Fanuc KAREL source: IO0072.KL

-- PROVISIONAL review KL for V940-1; original PC SHA256 c1c2a99b13fa0c8d7c35f1b90c9735473d2f50d53c25b610d3cd1d38be079865
-- Incomplete behavior may be omitted. Consult companion uncertainty JSON. Do not deploy.
PROGRAM IO0072
%NOLOCKGROUP
-- UNRESOLVED_LOCAL_POOL 5 cells at code offset 13; source declarations unknown
-- DIRECT_LOCAL_WORD_ACCESS alone does not prove INTEGER, REAL, or BOOLEAN
BEGIN
  -- V9_ZERO_TABLE_METADATA_HINT layout=0001; no indexed target words; source/name/runtime held
  -- V9_ZERO_GLOBAL_LAYOUT_HINT count-one $GROUP table, zero relocation slots, two routine descriptors; executable preamble and source held
  -- V9_ANALOG_RDI_SIGNAL_HINT AIN read I_plus_1
  -- UNRESOLVED_PC offsets 0-18; opcodes 2B,2C,7B
  -- UNRESOLVED_PC offsets 23-30; opcodes 9D,23
  -- UNRESOLVED_PC offsets 35-49; opcodes 2E,22,9D,33,35
  -- UNRESOLVED_PC offsets 54-61; opcodes 9D,23
  -- UNRESOLVED_PC offsets 66-77; opcodes 2E,23
  -- UNRESOLVED_PC offsets 82-99; opcodes 21,9D,52,19,64,23
  -- UNRESOLVED_PC offsets 104-108; opcodes 7F
  -- UNRESOLVED_PC offsets 113-117; opcodes 27,AA
  -- UNRESOLVED_PC offsets 122-126; opcodes 7F
END IO0072
